// TIA Portal V17 export
// export: Created 2024-06-16T17:47:30.7318914Z, ExportSetting WithDefaults, DisplayName Totally Integrated Automation Portal, DisplayVersion V17, DisplayName TIA Portal Openness, DisplayVersion V17, DisplayName TIA Portal Version Control Interface, DisplayVersion V17, DisplayName STEP 7 Professional, DisplayVersion V17, DisplayName STEP 7 Safety, DisplayVersion V17, DisplayName WinCC Professional, DisplayVersion V17
DATA_BLOCK "Obj_St3"   // DB300
VERSION : 0.1
// stored: AutoNumber false, DBAccessibleFromOPCUA true, DBAccessibleFromWebserver true, InstanceOfName Obj_St3_FB, InstanceOfType FB
"Obj_St3_FB"
   // VAR
   //    Axe_X1 : Struct
   //       _ActPos : Real;
   //       _ActVel : Real;
   //       _Mode : Int;
   //       Home : Bool;
   //       Halt : Bool;
   //       Jog : Bool;
   //       MoveAbs : Bool;
   //       MoveRel : Bool;
   //       MoveVel : Bool;
   //       PowerOff : Bool;
   //       PowerOn : Bool;
   //       SensPos : Bool;
   //       SensNeg : Bool;
   //       xBusy : Bool;
   //       xHomed : Bool;
   //       xMoveAbsDone : Bool;
   //       xMoveRelDone : Bool;
   //       xPower : Bool;
   //    END_STRUCT;
   //    Axe_X2 : Struct
   //       _ActPos : Real;
   //       _ActVel : Real;
   //       _Mode : Int;
   //       Home : Bool;
   //       Halt : Bool;
   //       Jog : Bool;
   //       MoveAbs : Bool;
   //       MoveRel : Bool;
   //       MoveVel : Bool;
   //       PowerOff : Bool;
   //       PowerOn : Bool;
   //       SensPos : Bool;
   //       SensNeg : Bool;
   //       xBusy : Bool;
   //       xHomed : Bool;
   //       xMoveAbsDone : Bool;
   //       xMoveRelDone : Bool;
   //       xPower : Bool;
   //    END_STRUCT;
   //    Axe_Y : Struct
   //       _ActPos : Real;
   //       _ActVel : Real;
   //       _Mode : Int;
   //       Home : Bool;
   //       Halt : Bool;
   //       Jog : Bool;
   //       MoveAbs : Bool;
   //       MoveRel : Bool;
   //       MoveVel : Bool;
   //       PowerOff : Bool;
   //       PowerOn : Bool;
   //       SensPos : Bool;
   //       SensNeg : Bool;
   //       xBusy : Bool;
   //       xHomed : Bool;
   //       xMoveAbsDone : Bool;
   //       xMoveRelDone : Bool;
   //       xPower : Bool;
   //    END_STRUCT;
   //    Axe_Z : Struct
   //       _ActPos : Real;
   //       _ActVel : Real;
   //       _Mode : Int;
   //       Home : Bool;
   //       Halt : Bool;
   //       Jog : Bool;
   //       MoveAbs : Bool;
   //       MoveRel : Bool;
   //       MoveVel : Bool;
   //       PowerOff : Bool;
   //       PowerOn : Bool;
   //       SensPos : Bool;
   //       SensNeg : Bool;
   //       xBusy : Bool;
   //       xHomed : Bool;
   //       xMoveAbsDone : Bool;
   //       xMoveRelDone : Bool;
   //       xPower : Bool;
   //    END_STRUCT;
   // END_VAR
BEGIN
END_DATA_BLOCK
